{attribute 'qualified_only'}
{attribute 'strict'}
TYPE E_Locations :
(
	MainPLC,
	MainPower_230V, 
	MainPower_24V, 
	MainAirSupply,
	MainScreen,
	MainIO,
	RemoteIO
);
END_TYPE

(* stored: Version 1.1.0.1, ProductVersion 3.1.4024.11
   EnumerationTextList E_Locations: Id {7410c5f4-a74b-47b1-9681-555f2dee9cf7} *)
